TYPE "Box"
VERSION : 0.1
   STRUCT
      min { S7_SetPoint := 'False'} : "Point";
      max { S7_SetPoint := 'False'} : "Point";
   END_STRUCT;

END_TYPE

